Yaskawa INFORM job: X2_6-7(-90,0).JBI

/JOB
//NAME X2_6-7(-90,0)
///FOLDERNAME X2
//POS
///NPOS 185,185,185,7,0,0
///TOOL 0
///POSTYPE PULSE
///PULSE
C00000=-2000,-52226,-115808,0,87402,0
C00001=123778,-52226,-115808,13625,87402,38668
C00002=121445,-23507,-59889,13798,60294,50612
C00003=120971,-19530,-53998,14347,58833,50249
C00004=120789,-17917,-51607,14569,58240,50101
C00005=120546,-14954,-49390,14716,58433,50037
C00006=120593,-15341,-49699,14684,58417,50052
C00007=120588,-15999,-48496,14856,57374,49905
C00008=120593,-15341,-49699,14684,58417,50052
C00009=121230,-20855,-58006,13919,60526,50564
C00010=121452,-23718,-59925,13805,60209,50604
C00011=120976,-19730,-54031,14355,58752,50240
C00012=120795,-18112,-51639,14578,58160,50092
C00013=120551,-15149,-49424,14724,58356,50028
C00014=120588,-15559,-49746,14700,58338,50040
C00015=120583,-16212,-48540,14873,57294,49892
C00016=120588,-15559,-49746,14700,58338,50040
C00017=121226,-21088,-58057,13934,60440,50552
C00018=80330,12074,-32837,40807,82496,30281
C00019=80327,10685,-31048,40947,81106,29736
C00020=80502,10915,-29678,40944,80476,29559
C00021=80494,10793,-29553,40959,80370,29517
C00022=80286,10450,-31099,40971,81055,29699
C00023=80289,11832,-32896,40829,82444,30245
C00024=123778,-52226,-115808,13625,87402,38668
C00025=86045,-26081,-114676,21990,103345,46267
C00026=1753,-99654,-106644,38855,72418,50846
C00027=11595,-142165,-93510,63811,60583,60768
C00028=145423,-153935,-109808,-60118,49898,-25166
C00029=129683,-14433,-46451,-37437,63836,-42675
C00030=126156,15994,-17969,-38339,57307,-41711
C00031=121195,61539,37577,-34493,60864,-29249
C00032=120895,68180,48215,-35390,58148,-28408
C00033=120778,71130,52879,-35829,56988,-28026
C00034=120620,75119,57652,-36096,56195,-27798
C00035=120650,74195,56504,-36020,56397,-27862
C00036=120646,74735,58827,-36470,55457,-27494
C00037=120650,74195,56504,-36020,56397,-27862
C00038=121059,64214,40619,-34587,60396,-29146
C00039=120400,59463,38509,-20824,46711,-38539
C00040=120723,68172,51850,-22428,43312,-37528
C00041=120780,69929,54520,-22775,42642,-37316
C00042=120621,73978,59351,-23030,41773,-37158
C00043=120650,73408,58633,-22989,41919,-37183
C00044=120647,74094,61137,-23515,40821,-36867
C00045=120650,73408,58633,-22989,41919,-37183
C00046=120390,73683,60474,-23221,40930,-37041
C00047=121275,74451,61405,-24003,41019,-36579
C00048=120390,73683,60474,-23221,40930,-37041
C00049=120002,62437,43371,-21025,45239,-38386
C00050=121727,63819,30741,-2584,89387,4744
C00051=121480,68384,39442,-2543,86374,4723
C00052=121383,70410,43182,-2529,85111,4717
C00053=121218,74045,47509,-2503,84311,4677
C00054=121254,73332,46624,-2508,84491,4686
C00055=121251,73438,48410,-2511,83447,4705
C00056=121254,73332,46624,-2508,84491,4686
C00057=119688,70398,44873,-2240,84015,4169
C00058=119612,72308,47140,-2229,83600,4150
C00059=120494,72941,47902,-2381,83482,4450
C00060=119612,72308,47140,-2229,83600,4150
C00061=119936,68722,40842,-2279,85639,4223
C00062=120898,67403,39050,-4403,76863,4671
C00063=120782,69888,43144,-4389,75618,4675
C00064=120624,73527,47467,-4356,74821,4649
C00065=120646,72661,46408,-4359,75029,4649
C00066=120642,72781,48210,-4378,73984,4685
C00067=120646,72661,46408,-4359,75029,4649
C00068=121054,64225,32391,-4413,79329,4636
C00069=119488,39968,14647,-36014,67920,-25782
C00070=118988,45247,23141,-36433,65662,-25200
C00071=111508,56039,27498,-17117,72177,-27375
C00072=112377,50002,21598,-8401,67422,-37537
C00073=118956,52577,24408,-9067,67547,-36073
C00074=127579,46805,22661,-29598,65663,-24889
C00075=127841,41491,14086,-29195,67986,-25419
C00076=124394,42362,3729,-9960,86928,6401
C00077=123788,46520,11118,-9812,84481,6397
C00078=123235,54024,19169,-9076,86584,6143
C00079=118293,52145,16987,-8931,87070,4312
C00080=117969,43371,7711,-8177,84334,4500
C00081=118453,39180,347,-8297,86736,4499
C00082=120386,37804,11026,-5111,57253,-30158
C00083=121449,41006,13740,-5776,57300,-29748
C00084=121390,46046,22695,-5937,54387,-29608
C00085=120149,57256,31234,-4750,62817,-30501
C00086=119721,38927,15273,-4805,55182,-30325
C00087=119005,37000,12159,-4298,56067,-30649
C00088=126156,15994,-17969,-38339,57307,-41711
C00089=129683,-14433,-46451,-37437,63836,-42675
C00090=145423,-153935,-109808,-60118,49898,-25166
C00091=118033,-154596,-109950,-60122,48986,-25325
C00092=23354,-154366,-109937,-60124,48858,-25410
C00093=-1117,-150372,-109058,-58139,47092,-27177
C00094=45296,29679,-47339,6439,84069,65831
C00095=121140,-42496,-73993,5628,49283,46430
C00096=120944,37759,2787,5314,56248,46752
C00097=120198,61864,38285,34319,60414,28991
C00098=120487,68617,49050,35242,57681,28141
C00099=120600,71949,53244,35522,56923,27907
C00100=120601,75012,56910,35777,56363,27693
C00101=120601,74293,56548,35833,56242,27647
C00102=120601,74581,57792,36074,55736,27451
C00103=120601,74293,56548,35833,56242,27647
C00104=120327,64556,41336,34416,59950,28887
C00105=120973,60901,35755,17710,55828,31005
C00106=120693,67769,46431,18542,52993,30375
C00107=121328,70625,50015,18330,52151,30497
C00108=121325,73378,53291,18480,51580,30387
C00109=121327,72516,52819,18517,51435,30360
C00110=121327,72743,53997,18671,50856,30247
C00111=121327,72516,52819,18517,51435,30360
C00112=120810,72505,52806,18836,51555,30152
C00113=120309,72509,52812,19145,51667,29951
C00114=120810,72505,52806,18836,51555,30152
C00115=121400,63688,40422,17755,54362,30929
C00116=119736,63940,30894,2141,88981,-4821
C00117=119969,68562,39652,2101,85963,-4794
C00118=120061,70613,43418,2088,84697,-4785
C00119=120066,73317,46630,2088,84108,-4791
C00120=120063,72481,45635,2088,84293,-4789
C00121=120063,72532,46608,2089,83720,-4797
C00122=120061,71563,44804,2088,84331,-4789
C00123=122084,70024,42982,1728,84613,-4108
C00124=122202,70062,43786,1707,84133,-4074
C00125=121433,70018,43734,1843,84160,-4333
C00126=122162,70059,43783,1714,84135,-4089
C00127=119736,63940,30894,2141,88981,-4821
C00128=120197,62152,30049,4056,79350,-4774
C00129=120486,67901,39637,4008,76396,-4773
C00130=120598,70419,43769,3994,75145,-4775
C00131=120758,74076,48115,3960,74343,-4746
C00132=120721,73217,47075,3967,74544,-4752
C00133=120718,73371,48919,3988,73491,-4787
C00134=120721,73217,47075,3967,74544,-4752
C00135=120327,64667,32928,4022,78865,-4747
C00136=120686,45927,23491,38955,63174,28378
C00137=120686,46108,26597,39536,61749,27794
C00138=120686,45934,26391,39524,61777,27806
C00139=120683,45149,23421,28756,58733,30420
C00140=120396,45326,23600,28776,58770,30351
C00141=120577,42139,18513,28267,60023,30784
C00142=120687,45991,21267,28124,60227,30888
C00143=120686,47026,12819,8567,83022,-5592
C00144=120687,47031,12825,8567,83022,-5592
C00145=120686,48013,14656,8577,82406,-5635
C00146=127376,44497,10084,6612,82803,-3406
C00147=120687,46974,12763,8567,83030,-5591
C00148=120686,46969,12758,8567,83031,-5592
C00149=120687,45951,18951,4057,57873,28006
C00150=120524,45585,19496,4178,57358,27923
C00151=120412,48146,23787,4310,56044,27828
C00152=121383,47898,25364,3760,54899,28172
C00153=120686,45853,22508,4160,55639,27920
C00154=120687,45855,20830,4111,56670,27961
C00155=120944,37759,2787,5314,56248,46752
C00156=121029,6109,-31455,5429,55754,46691
C00157=121124,-47303,-60190,6879,38381,45654
C00158=90302,-96069,-89343,23555,38901,42495
C00159=-3816,-1311,-64994,31572,95613,67531
C00160=70564,1634,-67433,11516,70070,68207
C00161=119867,-24433,-59136,-14152,58937,-50614
C00162=120397,-19684,-52272,-14797,57293,-50193
C00163=120506,-18656,-50780,-14937,56935,-50101
C00164=120511,-14672,-47812,-14905,57149,-50129
C00165=120710,-15025,-48128,-15045,57197,-50059
C00166=120710,-15355,-47467,-15140,56638,-49978
C00167=120710,-16128,-48956,-15054,57141,-50052
C00168=120091,-21825,-57337,-14276,59198,-50567
C00169=119857,-24210,-59144,-14128,59051,-50633
C00170=120415,-19213,-51898,-14807,57308,-50188
C00171=120495,-18452,-50792,-14911,57042,-50120
C00172=120497,-14821,-48084,-14881,57237,-50144
C00173=120721,-15441,-48584,-15042,57262,-50065
C00174=120721,-15856,-47752,-15161,56562,-49963
C00175=120721,-15884,-48916,-15045,57239,-50062
C00176=120103,-21564,-57292,-14269,59304,-50577
C00177=80258,11096,-32246,3966,63735,-54150
C00178=80233,9990,-30925,4031,62359,-54207
C00179=80616,11148,-28877,3798,61679,-54096
C00180=80987,12657,-27422,3557,61541,-53972
C00181=80296,10026,-30364,4000,62029,-54197
C00182=80299,11339,-32196,3936,63828,-54133
C00183=85671,813,-76116,-1319,91808,-19804
C00184=-2000,-87067,-95572,0,78525,0
BC00000=49710,523905,995172
BC00001=194136,440691,995172
BC00002=257010,445709,1075139
BC00003=257010,445709,1075139
BC00004=257010,445709,1075139
BC00005=257010,445709,1075139
BC00006=257010,445709,1075139
BC00007=257010,445709,1075139
BC00008=257010,445709,1075139
BC00009=257010,445709,1075139
BC00010=204484,436656,1075139
BC00011=204484,436656,1075139
BC00012=204484,436656,1075139
BC00013=204484,436656,1075139
BC00014=204484,436656,1075139
BC00015=204484,436656,1075139
BC00016=204484,436656,1075139
BC00017=204484,436656,1075139
BC00018=171955,446101,1075139
BC00019=172284,440665,1075139
BC00020=172415,438490,1075139
BC00021=105471,426943,1075139
BC00022=105340,429117,1075139
BC00023=105012,434554,1075139
BC00024=194136,440691,995172
BC00025=190418,454754,924402
BC00026=182211,485799,768176
BC00027=170886,523905,17
BC00028=170886,523905,17
BC00029=170886,523905,17
BC00030=170886,523905,17
BC00031=167868,515327,17
BC00032=167868,515327,17
BC00033=167868,515327,17
BC00034=167868,515327,17
BC00035=167868,515327,17
BC00036=167868,515327,17
BC00037=167868,515327,17
BC00038=167868,515327,17
BC00039=156913,523889,17
BC00040=156913,523889,17
BC00041=156913,523889,17
BC00042=156913,523889,17
BC00043=156913,523889,17
BC00044=156913,523889,17
BC00045=156913,523889,17
BC00046=156913,523889,17
BC00047=156913,523889,17
BC00048=156913,523889,17
BC00049=156913,523889,17
BC00050=165442,473316,64867
BC00051=165442,473316,64867
BC00052=165442,473316,64867
BC00053=165442,473316,64867
BC00054=165442,473316,64867
BC00055=165442,473316,64867
BC00056=165442,473316,64867
BC00057=165442,473316,64867
BC00058=165442,473316,64867
BC00059=165442,473316,64867
BC00060=165442,473316,64867
BC00061=165442,473316,64867
BC00062=146162,487166,44203
BC00063=146162,487166,44203
BC00064=146162,487166,44203
BC00065=146162,487166,44203
BC00066=146162,487166,44203
BC00067=146162,487166,44203
BC00068=146162,487166,44203
BC00069=161236,484900,17
BC00070=161236,484900,17
BC00071=161236,484900,17
BC00072=161236,484900,17
BC00073=161236,484900,17
BC00074=161236,484900,17
BC00075=161236,484900,17
BC00076=144204,461025,3501
BC00077=144204,461025,3501
BC00078=144204,461025,3501
BC00079=144204,461025,3501
BC00080=144204,461025,3501
BC00081=144204,461025,3501
BC00082=173416,495229,17
BC00083=173416,495229,17
BC00084=173416,495229,17
BC00085=173415,495229,15
BC00086=173416,495229,17
BC00087=173416,495229,17
BC00088=170886,523905,17
BC00089=170886,523905,17
BC00090=170886,523905,17
BC00091=170886,523905,17
BC00092=170886,523905,17
BC00093=170886,523905,1054911
BC00094=180654,582681,422088
BC00095=268409,523905,17
BC00096=268409,523905,17
BC00097=270577,513971,17
BC00098=270577,513971,17
BC00099=270576,513971,14
BC00100=270576,513971,14
BC00101=270576,513971,14
BC00102=270576,513971,14
BC00103=270576,513971,14
BC00104=270577,513971,17
BC00105=281347,515946,17
BC00106=281347,515946,17
BC00107=281347,515946,17
BC00108=281347,515946,17
BC00109=281347,515946,17
BC00110=281347,515946,17
BC00111=281347,515946,17
BC00112=281347,515946,17
BC00113=281347,515946,17
BC00114=281347,515946,17
BC00115=281347,515946,17
BC00116=271605,472778,62085
BC00117=271605,472778,62085
BC00118=271605,472778,62085
BC00119=271605,472778,62085
BC00120=271605,472778,62085
BC00121=271605,472778,62085
BC00122=271605,472778,62085
BC00123=271605,472778,62085
BC00124=271605,472778,62085
BC00125=271605,472778,62085
BC00126=271605,472778,62085
BC00127=271605,472778,62085
BC00128=291338,486602,41666
BC00129=291338,486602,41666
BC00130=291338,486602,41666
BC00131=291338,486602,41666
BC00132=291338,486602,41666
BC00133=291338,486602,41666
BC00134=291338,486602,41666
BC00135=291338,486602,41666
BC00136=274613,493094,17
BC00137=272953,487860,17
BC00138=272402,486124,17
BC00139=262519,491641,17
BC00140=297522,485598,16
BC00141=298630,486167,16
BC00142=301037,492725,17
BC00143=304994,466183,27741
BC00144=303333,460949,8883
BC00145=302996,459885,5051
BC00146=302997,459886,5049
BC00147=284698,464197,8574
BC00148=286358,469431,27433
BC00149=262606,499983,17
BC00150=262225,495040,17
BC00151=262225,495040,17
BC00152=262033,495223,17
BC00153=259916,496527,17
BC00154=258338,500710,17
BC00155=268409,523905,17
BC00156=268409,523905,17
BC00157=268409,523905,17
BC00158=228111,523069,176209
BC00159=26262,518880,1058751
BC00160=125635,474792,1068548
BC00161=180197,447562,1075139
BC00162=180197,447562,1075139
BC00163=180197,447562,1075139
BC00164=180197,447562,1075139
BC00165=180197,447562,1075139
BC00166=180197,447562,1075139
BC00167=180197,447562,1075139
BC00168=180197,447562,1075139
BC00169=234485,438072,1075139
BC00170=234485,438072,1075139
BC00171=234485,438072,1075139
BC00172=234485,438072,1075139
BC00173=234485,438072,1075139
BC00174=234485,438072,1075139
BC00175=234485,438072,1075139
BC00176=234485,438072,1075139
BC00177=58212,448278,1075139
BC00178=57851,441575,1075139
BC00179=57799,440617,1075139
BC00180=124839,431145,1075139
BC00181=124839,431145,1075139
BC00182=125134,436617,1075139
BC00183=180828,447635,1075139
BC00184=66564,515818,1075139
EC00000=798156,-183832
EC00001=798156,-183832
EC00002=798156,-183832
EC00003=798156,-183832
EC00004=798156,-183832
EC00005=798156,-183832
EC00006=798156,-183832
EC00007=798156,-183832
EC00008=798156,-183832
EC00009=798156,-183832
EC00010=798156,-183832
EC00011=798156,-183832
EC00012=798156,-183832
EC00013=798156,-183832
EC00014=798156,-183832
EC00015=798156,-183832
EC00016=798156,-183832
EC00017=798156,-183832
EC00018=798156,-183832
EC00019=798156,-183832
EC00020=798156,-183832
EC00021=798156,-183832
EC00022=798156,-183832
EC00023=798156,-183832
EC00024=798156,-183832
EC00025=798156,-183832
EC00026=798156,-183832
EC00027=798156,-183832
EC00028=798156,-183832
EC00029=798156,-183832
EC00030=798156,-183832
EC00031=798156,-183832
EC00032=798156,-183832
EC00033=798156,-183832
EC00034=798156,-183832
EC00035=798156,-183832
EC00036=798156,-183832
EC00037=798156,-183832
EC00038=798156,-183832
EC00039=798156,-183832
EC00040=798156,-183832
EC00041=798156,-183832
EC00042=798156,-183832
EC00043=798156,-183832
EC00044=798156,-183832
EC00045=798156,-183832
EC00046=798156,-183832
EC00047=798156,-183832
EC00048=798156,-183832
EC00049=798156,-183832
EC00050=798156,-183832
EC00051=798156,-183832
EC00052=798156,-183832
EC00053=798156,-183832
EC00054=798156,-183832
EC00055=798156,-183832
EC00056=798156,-183832
EC00057=798156,-183832
EC00058=798156,-183832
EC00059=798156,-183832
EC00060=798156,-183832
EC00061=798156,-183832
EC00062=798156,-183832
EC00063=798156,-183832
EC00064=798156,-183832
EC00065=798156,-183832
EC00066=798156,-183832
EC00067=798156,-183832
EC00068=798156,-183832
EC00069=798156,-183832
EC00070=798156,-183832
EC00071=798156,-183832
EC00072=798156,-183832
EC00073=798156,-183832
EC00074=798156,-183832
EC00075=798156,-183832
EC00076=798156,-183832
EC00077=798156,-183832
EC00078=798156,-183832
EC00079=798156,-183832
EC00080=798156,-183832
EC00081=798156,-183832
EC00082=798156,-183832
EC00083=798156,-183832
EC00084=798156,-183832
EC00085=798155,-183832
EC00086=798156,-183832
EC00087=798156,-183832
EC00088=798156,-183832
EC00089=798156,-183832
EC00090=798156,-183832
EC00091=878342,-390207
EC00092=878342,-1035719
EC00093=798156,-1296783
EC00094=798156,-1296783
EC00095=798156,-1296783
EC00096=798156,-1296783
EC00097=798156,-1296783
EC00098=798156,-1296783
EC00099=798155,-1296783
EC00100=798155,-1296783
EC00101=798155,-1296783
EC00102=798155,-1296783
EC00103=798155,-1296783
EC00104=798156,-1296783
EC00105=798156,-1296783
EC00106=798156,-1296783
EC00107=798156,-1296783
EC00108=798156,-1296783
EC00109=798156,-1296783
EC00110=798156,-1296783
EC00111=798156,-1296783
EC00112=798156,-1296783
EC00113=798156,-1296783
EC00114=798156,-1296783
EC00115=798156,-1296783
EC00116=798156,-1296783
EC00117=798156,-1296783
EC00118=798156,-1296783
EC00119=798156,-1296783
EC00120=798156,-1296783
EC00121=798156,-1296783
EC00122=798156,-1296783
EC00123=798156,-1296783
EC00124=798156,-1296783
EC00125=798156,-1296783
EC00126=798156,-1296783
EC00127=798156,-1296783
EC00128=798156,-1296783
EC00129=798156,-1296783
EC00130=798156,-1296783
EC00131=798156,-1296783
EC00132=798156,-1296783
EC00133=798156,-1296783
EC00134=798156,-1296783
EC00135=798156,-1296783
EC00136=798156,-1296783
EC00137=798156,-1296783
EC00138=798156,-1296783
EC00139=798156,-1296783
EC00140=798155,-1296783
EC00141=798155,-1296783
EC00142=798156,-1296783
EC00143=798156,-1296783
EC00144=798156,-1296783
EC00145=798156,-1296783
EC00146=798155,-1296784
EC00147=798156,-1296783
EC00148=798156,-1296783
EC00149=798156,-1296783
EC00150=798156,-1296783
EC00151=798156,-1296783
EC00152=798156,-1296783
EC00153=798156,-1296783
EC00154=798156,-1296783
EC00155=798156,-1296783
EC00156=798156,-1296783
EC00157=798156,-1296783
EC00158=798156,-1296783
EC00159=798156,-1296783
EC00160=798156,-1296783
EC00161=798156,-1296783
EC00162=798156,-1296783
EC00163=798156,-1296783
EC00164=798156,-1296783
EC00165=798156,-1296783
EC00166=798156,-1296783
EC00167=798156,-1296783
EC00168=798156,-1296783
EC00169=798156,-1296783
EC00170=798156,-1296783
EC00171=798156,-1296783
EC00172=798156,-1296783
EC00173=798156,-1296783
EC00174=798156,-1296783
EC00175=798156,-1296783
EC00176=798156,-1296783
EC00177=798156,-1296783
EC00178=798156,-1296783
EC00179=798156,-1296783
EC00180=798156,-1296783
EC00181=798156,-1296783
EC00182=798156,-1296783
EC00183=798156,-1296783
EC00184=798156,-1296783
///POSTYPE BASE
///RECTAN
///RCONF 0,0,0,0,1,0,0,0,0,0,0,0,0,0,0,0,0,0,0,0,0,0,0,0
P00006=2.006,1.622,-0.565,0.0000,0.0000,0.0000
P00021=0.073,2.058,-0.109,0.0000,0.0000,0.0000
P00022=2.006,1.622,-0.565,0.0000,0.0000,0.0000
///RCONF 0,0,0,0,0,0,0,0,0,0,0,0,0,0,0,0,0,0,0,0,0,0,0,0
P00023=-2.957,-4.083,2.762,0.0000,0.0000,0.0000
P00024=-1.466,-0.226,-0.419,0.0000,0.0000,0.0000
P00025=3.643,0.007,-2.585,0.0000,0.0000,0.0000
P00026=2.644,0.055,-2.583,0.0000,0.0000,0.0000
//INST
///DATE 2024/11/27 09:27
///ATTR SC,RW
///GROUP1 RB1,BS1
///GROUP2 ST1
NOP
'X2_6-7(-90,0)
'Spoina W6
MOVJ C00000 BC00000 VJ=100.00  +MOVJ EC00000 VJ=100.00
MOVJ C00001 BC00001 VJ=100.00  +MOVJ EC00001 VJ=100.00
'Path S3970
SFTOF3D
MOVJ C00002 BC00002 VJ=100.00  +MOVJ EC00002 VJ=100.00
MOVL C00003 BC00003 V=666.7  +MOVJ EC00003 VJ=100.00
SMOVL C00004 BC00004 V=166.7  +MOVJ EC00004
SREFP 3 C00005 BC00005  +REFP EC00005
CALL JOB:SEARCH-R1-S13D
SET P021 P006
SFTON3D P021
SMOVL C00006 BC00006 V=166.7  +MOVJ EC00006
SREFP 3 C00007 BC00007  +REFP EC00007
CALL JOB:SEARCH-R1-S13D
SET P021 P006
SFTON3D P021
SMOVL C00008 BC00008 V=166.7  +MOVJ EC00008
MOVL C00009 BC00009 V=1000.0  +MOVJ EC00009 VJ=100.00
'EndPath S3970
'Path S3971
SFTOF3D
MOVJ C00010 BC00010 VJ=100.00  +MOVJ EC00010 VJ=100.00
MOVL C00011 BC00011 V=666.7  +MOVJ EC00011 VJ=100.00
SMOVL C00012 BC00012 V=166.7  +MOVJ EC00012
SREFP 3 C00013 BC00013  +REFP EC00013
CALL JOB:SEARCH-R1-S13D
SET P022 P006
SFTON3D P022
SMOVL C00014 BC00014 V=166.7  +MOVJ EC00014
SREFP 3 C00015 BC00015  +REFP EC00015
CALL JOB:SEARCH-R1-S13D
SET P022 P006
SFTON3D P022
SMOVL C00016 BC00016 V=166.7  +MOVJ EC00016
MOVL C00017 BC00017 V=1000.0  +MOVJ EC00017 VJ=100.00
'EndPath S3971
'Path W4862
SFTOF3D
SFTON3D P021
MOVJ C00018 BC00018 VJ=100.00  +MOVJ EC00018 VJ=100.00
SMOVL C00019 BC00019 V=666.7  +MOVJ EC00019
SMOVL C00020 BC00020 V=166.7 PL=0  +MOVJ EC00020
MACRO1 MJ#(0) ARGF14
ARCON
SFTON3D P022
SMOVL C00021 BC00021 V=10.0  +MOVJ EC00021
ARCOF
SMOVL C00022 BC00022 V=800.0  +MOVJ EC00022
SMOVL C00023 BC00023 V=1000.0  +MOVJ EC00023
SFTOF3D
'EndPath W4862
MOVJ C00024 BC00024 VJ=100.00  +MOVJ EC00024 VJ=100.00
MOVJ C00025 BC00025 VJ=100.00  +MOVJ EC00025 VJ=100.00
MOVJ C00026 BC00026 VJ=100.00  +MOVJ EC00026 VJ=100.00
CALL JOB:CLEAN-R1_KM_NEW
MOVJ C00027 BC00027 VJ=100.00  +MOVJ EC00027 VJ=100.00
MOVJ C00028 BC00028 VJ=100.00  +MOVJ EC00028 VJ=100.00
MOVJ C00029 BC00029 VJ=100.00  +MOVJ EC00029 VJ=100.00
MOVJ C00030 BC00030 VJ=100.00  +MOVJ EC00030 VJ=100.00
'Path S3972
SFTOF3D
MOVJ C00031 BC00031 VJ=100.00  +MOVJ EC00031 VJ=100.00
MOVL C00032 BC00032 V=666.7  +MOVJ EC00032 VJ=100.00
SMOVL C00033 BC00033 V=166.7  +MOVJ EC00033
SREFP 3 C00034 BC00034  +REFP EC00034
CALL JOB:SEARCH-R1-S13D
SET P023 P006
SFTON3D P023
SMOVL C00035 BC00035 V=166.7  +MOVJ EC00035
SREFP 3 C00036 BC00036  +REFP EC00036
CALL JOB:SEARCH-R1-S13D
SET P023 P006
SFTON3D P023
SMOVL C00037 BC00037 V=166.7  +MOVJ EC00037
MOVL C00038 BC00038 V=1000.0  +MOVJ EC00038 VJ=100.00
'EndPath S3972
'Path S3973
SFTOF3D
MOVJ C00039 BC00039 VJ=100.00  +MOVJ EC00039 VJ=100.00
MOVL C00040 BC00040 V=666.7  +MOVJ EC00040 VJ=100.00
SMOVL C00041 BC00041 V=166.7  +MOVJ EC00041
SREFP 3 C00042 BC00042  +REFP EC00042
CALL JOB:SEARCH-R1-S13D
SET P024 P006
SFTON3D P024
SMOVL C00043 BC00043 V=166.7  +MOVJ EC00043
SREFP 3 C00044 BC00044  +REFP EC00044
CALL JOB:SEARCH-R1-S13D
SET P024 P006
SFTON3D P024
SMOVL C00045 BC00045 V=166.7  +MOVJ EC00045
SMOVL C00046 BC00046 V=166.7  +MOVJ EC00046
SREFP 3 C00047 BC00047  +REFP EC00047
CALL JOB:SEARCH-R1-S13D
SET P024 P006
SFTON3D P024
SMOVL C00048 BC00048 V=166.7  +MOVJ EC00048
MOVL C00049 BC00049 V=1000.0  +MOVJ EC00049 VJ=100.00
'EndPath S3973
'Path S3974
SFTOF3D
MOVJ C00050 BC00050 VJ=100.00  +MOVJ EC00050 VJ=100.00
MOVL C00051 BC00051 V=666.7  +MOVJ EC00051 VJ=100.00
SMOVL C00052 BC00052 V=166.7  +MOVJ EC00052
SREFP 3 C00053 BC00053  +REFP EC00053
CALL JOB:SEARCH-R1-S13D
SET P025 P006
SFTON3D P025
SMOVL C00054 BC00054 V=166.7  +MOVJ EC00054
SREFP 3 C00055 BC00055  +REFP EC00055
CALL JOB:SEARCH-R1-S13D
SET P025 P006
SFTON3D P025
SMOVL C00056 BC00056 V=166.7  +MOVJ EC00056
SMOVL C00057 BC00057 V=166.7  +MOVJ EC00057
SMOVL C00058 BC00058 V=166.7  +MOVJ EC00058
SREFP 3 C00059 BC00059  +REFP EC00059
CALL JOB:SEARCH-R1-S13D
SET P025 P006
SFTON3D P025
SMOVL C00060 BC00060 V=166.7  +MOVJ EC00060
SMOVL C00061 BC00061 V=333.3  +MOVJ EC00061
'EndPath S3974
'Path S3975
SFTOF3D
MOVL C00062 BC00062 V=1000.0  +MOVJ EC00062 VJ=100.00
SMOVL C00063 BC00063 V=166.7  +MOVJ EC00063
SREFP 3 C00064 BC00064  +REFP EC00064
CALL JOB:SEARCH-R1-S13D
SET P026 P006
SFTON3D P026
SMOVL C00065 BC00065 V=166.7  +MOVJ EC00065
SREFP 3 C00066 BC00066  +REFP EC00066
CALL JOB:SEARCH-R1-S13D
SET P026 P006
SFTON3D P026
SMOVL C00067 BC00067 V=166.7  +MOVJ EC00067
MOVL C00068 BC00068 V=1000.0  +MOVJ EC00068 VJ=100.00
'EndPath S3975
'Path W3973
SFTOF3D
SFTON3D P023
MOVJ C00069 BC00069 VJ=100.00  +MOVJ EC00069 VJ=100.00
SMOVL C00070 BC00070 V=800.0  +MOVJ EC00070
SMOVL C00071 BC00071 V=150.0 PL=0  +MOVJ EC00071
ARCON
SMOVL C00072 BC00072 V=10.5  +MOVJ EC00072
SFTON3D P024
SMOVL C00073 BC00073 V=10.5  +MOVJ EC00073
ARCOF
SMOVL C00074 BC00074 V=800.0  +MOVJ EC00074
SMOVL C00075 BC00075 V=1000.0  +MOVJ EC00075
SFTOF3D
'EndPath W3973
'Path W3976
SFTOF3D
SFTON3D P026
MOVJ C00076 BC00076 VJ=100.00  +MOVJ EC00076 VJ=100.00
SMOVL C00077 BC00077 V=800.0  +MOVJ EC00077
SMOVL C00078 BC00078 V=150.0 PL=0  +MOVJ EC00078
ARCON
SFTON3D P025
SMOVL C00079 BC00079 V=10.5  +MOVJ EC00079
ARCOF
SMOVL C00080 BC00080 V=800.0  +MOVJ EC00080
SMOVL C00081 BC00081 V=1000.0  +MOVJ EC00081
SFTOF3D
'EndPath W3976
'Path W3977
SFTOF3D
SFTON3D P025
MOVJ C00082 BC00082 VJ=100.00  +MOVJ EC00082 VJ=100.00
SMOVL C00083 BC00083 V=800.0  +MOVJ EC00083
SMOVL C00084 BC00084 V=150.0 PL=0  +MOVJ EC00084
ARCON
SFTON3D P024
SMOVL C00085 BC00085 V=11.7  +MOVJ EC00085
ARCOF
SMOVL C00086 BC00086 V=800.0  +MOVJ EC00086
SMOVL C00087 BC00087 V=1000.0  +MOVJ EC00087
SFTOF3D
'EndPath W3977
MOVJ C00088 BC00088 VJ=100.00  +MOVJ EC00088 VJ=100.00
MOVJ C00089 BC00089 VJ=100.00  +MOVJ EC00089 VJ=100.00
MOVJ C00090 BC00090 VJ=100.00  +MOVJ EC00090 VJ=100.00
MOVJ C00091 BC00091 VJ=100.00  +MOVJ EC00091 VJ=100.00
MOVJ C00092 BC00092 VJ=100.00  +MOVJ EC00092 VJ=100.00
MOVJ C00093 BC00093 VJ=100.00  +MOVJ EC00093 VJ=100.00
'wire_cut
CALL JOB:CLEAN-R1_KM_NEW
'wire_cut
MOVJ C00094 BC00094 VJ=50.00  +MOVJ EC00094 VJ=50.00
MOVJ C00095 BC00095 VJ=100.00  +MOVJ EC00095 VJ=100.00
MOVJ C00096 BC00096 VJ=100.00  +MOVJ EC00096 VJ=100.00
'Spoina W7
'Path S3987
SFTOF3D
MOVJ C00097 BC00097 VJ=100.00  +MOVJ EC00097 VJ=100.00
MOVL C00098 BC00098 V=666.7  +MOVJ EC00098 VJ=100.00
SMOVL C00099 BC00099 V=166.7  +MOVJ EC00099
SREFP 3 C00100 BC00100  +REFP EC00100
CALL JOB:SEARCH-R1-S13D
SET P023 P006
SFTON3D P023
SMOVL C00101 BC00101 V=166.7  +MOVJ EC00101
SREFP 3 C00102 BC00102  +REFP EC00102
CALL JOB:SEARCH-R1-S13D
SET P023 P006
SFTON3D P023
SMOVL C00103 BC00103 V=166.7  +MOVJ EC00103
MOVL C00104 BC00104 V=1000.0  +MOVJ EC00104 VJ=100.00
'EndPath S3987
'Path S3988
SFTOF3D
MOVJ C00105 BC00105 VJ=100.00  +MOVJ EC00105 VJ=100.00
MOVL C00106 BC00106 V=666.7  +MOVJ EC00106 VJ=100.00
SMOVL C00107 BC00107 V=166.7  +MOVJ EC00107
SREFP 3 C00108 BC00108  +REFP EC00108
CALL JOB:SEARCH-R1-S13D
SET P024 P006
SFTON3D P024
SMOVL C00109 BC00109 V=166.7  +MOVJ EC00109
SREFP 3 C00110 BC00110  +REFP EC00110
CALL JOB:SEARCH-R1-S13D
SET P024 P006
SFTON3D P024
SMOVL C00111 BC00111 V=166.7  +MOVJ EC00111
SMOVL C00112 BC00112 V=166.7  +MOVJ EC00112
SREFP 3 C00113 BC00113  +REFP EC00113
CALL JOB:SEARCH-R1-S13D
SET P024 P006
SFTON3D P024
SMOVL C00114 BC00114 V=166.7  +MOVJ EC00114
MOVL C00115 BC00115 V=1000.0  +MOVJ EC00115 VJ=100.00
'EndPath S3988
'Path S3989
SFTOF3D
MOVJ C00116 BC00116 VJ=100.00  +MOVJ EC00116 VJ=100.00
MOVL C00117 BC00117 V=666.7  +MOVJ EC00117 VJ=100.00
SMOVL C00118 BC00118 V=166.7  +MOVJ EC00118
SREFP 3 C00119 BC00119  +REFP EC00119
CALL JOB:SEARCH-R1-S13D
SET P025 P006
SFTON3D P025
SMOVL C00120 BC00120 V=166.7  +MOVJ EC00120
SREFP 3 C00121 BC00121  +REFP EC00121
CALL JOB:SEARCH-R1-S13D
SET P025 P006
SFTON3D P025
SMOVL C00122 BC00122 V=166.7  +MOVJ EC00122
SMOVL C00123 BC00123 V=333.3  +MOVJ EC00123
SMOVL C00124 BC00124 V=166.7  +MOVJ EC00124
SREFP 3 C00125 BC00125  +REFP EC00125
CALL JOB:SEARCH-R1-S13D
SET P025 P006
SFTON3D P025
SMOVL C00126 BC00126 V=166.7  +MOVJ EC00126
MOVL C00127 BC00127 V=1000.0  +MOVJ EC00127 VJ=100.00
'EndPath S3989
'Path S3990
SFTOF3D
MOVJ C00128 BC00128 VJ=100.00  +MOVJ EC00128 VJ=100.00
MOVL C00129 BC00129 V=666.7  +MOVJ EC00129 VJ=100.00
SMOVL C00130 BC00130 V=166.7  +MOVJ EC00130
SREFP 3 C00131 BC00131  +REFP EC00131
CALL JOB:SEARCH-R1-S13D
SET P026 P006
SFTON3D P026
SMOVL C00132 BC00132 V=166.7  +MOVJ EC00132
SREFP 3 C00133 BC00133  +REFP EC00133
CALL JOB:SEARCH-R1-S13D
SET P026 P006
SFTON3D P026
SMOVL C00134 BC00134 V=166.7  +MOVJ EC00134
MOVL C00135 BC00135 V=1000.0  +MOVJ EC00135 VJ=100.00
'EndPath S3990
'Path W3991
SFTOF3D
SFTON3D P023
MOVJ C00136 BC00136 VJ=100.00  +MOVJ EC00136 VJ=100.00
SMOVL C00137 BC00137 V=666.7  +MOVJ EC00137
SMOVL C00138 BC00138 V=150.0 PL=0  +MOVJ EC00138
ARCON
SMOVL C00139 BC00139 V=10.8  +MOVJ EC00139
SFTON3D P024
SMOVL C00140 BC00140 V=10.8  +MOVJ EC00140
ARCOF
SMOVL C00141 BC00141 V=800.0  +MOVJ EC00141
SMOVL C00142 BC00142 V=1000.0  +MOVJ EC00142
SFTOF3D
'EndPath W3991
'Path W3992
SFTOF3D
SFTON3D P026
MOVJ C00143 BC00143 VJ=100.00  +MOVJ EC00143 VJ=100.00
SMOVL C00144 BC00144 V=800.0  +MOVJ EC00144
SMOVL C00145 BC00145 V=150.0 PL=0  +MOVJ EC00145
ARCON
SFTON3D P025
SMOVL C00146 BC00146 V=10.8  +MOVJ EC00146
ARCOF
SMOVL C00147 BC00147 V=800.0  +MOVJ EC00147
SMOVL C00148 BC00148 V=1000.0  +MOVJ EC00148
SFTOF3D
'EndPath W3992
'Path W3993
SFTOF3D
SFTON3D P025
MOVJ C00149 BC00149 VJ=100.00  +MOVJ EC00149 VJ=100.00
SMOVL C00150 BC00150 V=800.0  +MOVJ EC00150
SMOVL C00151 BC00151 V=150.0 PL=0  +MOVJ EC00151
ARCON
SFTON3D P024
SMOVL C00152 BC00152 V=10.0  +MOVJ EC00152
ARCOF
SMOVL C00153 BC00153 V=800.0  +MOVJ EC00153
SMOVL C00154 BC00154 V=1000.0  +MOVJ EC00154
SFTOF3D
'EndPath W3993
'wire_cut
MOVJ C00155 BC00155 VJ=100.00  +MOVJ EC00155 VJ=100.00
MOVJ C00156 BC00156 VJ=100.00  +MOVJ EC00156 VJ=100.00
MOVJ C00157 BC00157 VJ=100.00  +MOVJ EC00157 VJ=100.00
MOVJ C00158 BC00158 VJ=100.00  +MOVJ EC00158 VJ=0.78
CALL JOB:CLEAN-R1_KM_NEW
MOVJ C00159 BC00159 VJ=100.00  +MOVJ EC00159 VJ=100.00
MOVJ C00160 BC00160 VJ=100.00  +MOVJ EC00160 VJ=100.00
'Path S3984
SFTOF3D
MOVJ C00161 BC00161 VJ=100.00  +MOVJ EC00161 VJ=100.00
MOVL C00162 BC00162 V=666.7  +MOVJ EC00162 VJ=100.00
SMOVL C00163 BC00163 V=166.7  +MOVJ EC00163
SREFP 3 C00164 BC00164  +REFP EC00164
CALL JOB:SEARCH-R1-S13D
SET P021 P006
SFTON3D P021
SMOVL C00165 BC00165 V=166.7  +MOVJ EC00165
SREFP 3 C00166 BC00166  +REFP EC00166
CALL JOB:SEARCH-R1-S13D
SET P021 P006
SFTON3D P021
SMOVL C00167 BC00167 V=166.7  +MOVJ EC00167
MOVL C00168 BC00168 V=1000.0  +MOVJ EC00168 VJ=100.00
'EndPath S3984
'Path S3985
SFTOF3D
MOVJ C00169 BC00169 VJ=100.00  +MOVJ EC00169 VJ=100.00
MOVL C00170 BC00170 V=666.7  +MOVJ EC00170 VJ=100.00
SMOVL C00171 BC00171 V=166.7  +MOVJ EC00171
SREFP 3 C00172 BC00172  +REFP EC00172
CALL JOB:SEARCH-R1-S13D
SET P022 P006
SFTON3D P022
SMOVL C00173 BC00173 V=166.7  +MOVJ EC00173
SREFP 3 C00174 BC00174  +REFP EC00174
CALL JOB:SEARCH-R1-S13D
SET P022 P006
SFTON3D P022
SMOVL C00175 BC00175 V=166.7  +MOVJ EC00175
MOVL C00176 BC00176 V=1000.0  +MOVJ EC00176 VJ=100.00
'EndPath S3985
'Path W4220
SFTOF3D
SFTON3D P021
MOVJ C00177 BC00177 VJ=100.00  +MOVJ EC00177 VJ=100.00
SMOVL C00178 BC00178 V=666.7  +MOVJ EC00178
SMOVL C00179 BC00179 V=150.0 PL=0  +MOVJ EC00179
ARCON
SFTON3D P022
SMOVL C00180 BC00180 V=10.0  +MOVJ EC00180
ARCOF
SMOVL C00181 BC00181 V=800.0  +MOVJ EC00181
SMOVL C00182 BC00182 V=1000.0  +MOVJ EC00182
SFTOF3D
'EndPath W4220
MOVJ C00183 BC00183 VJ=100.00  +MOVJ EC00183 VJ=100.00
MOVJ C00184 BC00184 VJ=100.00  +MOVJ EC00184 VJ=100.00
END
